FUNCTION_BLOCK ASRT_3AE_TO_SRT (* Composite FB for convert 3 AE to ASRT *)
  (* Standard: 61499-2; Description: Copyright (c) 2026 HR Agrartechnik GmbH This program and the accompanying materials are made available under the terms of the Eclipse Public License 2.0 which is available at https://www.eclipse.org/legal/epl-2.0/ SPDX-License-Identifier: EPL-2.0 *)
  (* Version 1.0, 2026-09-06, Franz Höpfinger, HR Agrartechnik GmbH *)
  PACKAGE adapter::conversion::unidirectional;
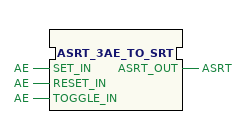
  SOCKETS
    SET_IN : adapter::types::unidirectional::AE; (* Set / Switch on *)
    RESET_IN : adapter::types::unidirectional::AE; (* Reset / Switch off *)
    TOGGLE_IN : adapter::types::unidirectional::AE; (* Toggle / Switch output *)
  END_SOCKETS
  PLUGS
    ASRT_OUT : adapter::types::unidirectional::ASRT; (* Adapter Output *)
  END_PLUGS
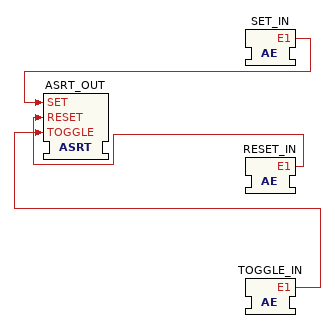
  EVENT_CONNECTIONS
    SET_IN.E1 TO ASRT_OUT.SET;
    RESET_IN.E1 TO ASRT_OUT.RESET;
    TOGGLE_IN.E1 TO ASRT_OUT.TOGGLE;
  END_CONNECTIONS
END_FUNCTION_BLOCK
